// TIA Portal V18 export
DATA_BLOCK "Interlocks_DB"   // DB3
VERSION : 0.1
// stored: AutoNumber true, InstanceOfName Interlocks_And_Permissive, InstanceOfType FB
"Interlocks_And_Permissive"
   // VAR_INPUT
   //    capacitive_HLS : Bool;
   //    temperature : Int;
   //    emergency_state : Bool;
   //    FCV_valve_closed : Bool;
   //    ESD_valve_closed : Bool;
   //    grounding : Bool;
   //    Temperature_threshold : Int;
   // END_VAR
   // VAR_OUTPUT
   //    interlocks_idle : Bool;
   //    interlocks_loading : Bool;
   // END_VAR
   // VAR
   //    Temperature_is_ok : Bool;
   // END_VAR
BEGIN
END_DATA_BLOCK
